// TIA Portal project "MaquinaEmbalarAut" (V14)
// Automated Packaging Machine Using PLC

(* hardware
DEVICE "S7-1200 station_1"  S7-1200 Station
   slot 0: "Rack_0"  S7-1200 Rack  Rack  V1.0
   slot 1: "Embaladora automatica"  CPU 1214C DC/DC/DC  6ES7 214-1AG40-0XB0  V4.2
*)

// ===== PLC "Embaladora automatica"  CPU 1214C DC/DC/DC =====

VAR_GLOBAL   // PLC tag table "Default tag table"
   "System_Byte" AT %MB0 : Byte;
   "FirstScan" AT %M0.0 : Bool;
   "DiagStatusUpdate" AT %M0.1 : Bool;
   "AlwaysTRUE" AT %M0.2 : Bool;
   "AlwaysFALSE" AT %M0.3 : Bool;
   "Clock_Byte" AT %MB1 : Byte;
   "Clock_10Hz" AT %M1.0 : Bool;
   "Clock_5Hz" AT %M1.1 : Bool;
   "Clock_2.5Hz" AT %M1.2 : Bool;
   "Clock_2Hz" AT %M1.3 : Bool;
   "Clock_1.25Hz" AT %M1.4 : Bool;
   "Clock_1Hz" AT %M1.5 : Bool;
   "Clock_0.625Hz" AT %M1.6 : Bool;
   "Clock_0.5Hz" AT %M1.7 : Bool;
   "LigaEsteiraCaixa" AT %M10.0 : Bool;
   "LigaEsteiraProdutos" AT %M20.0 : Bool;
   "Zera cont" AT %M100.5 : Bool;
END_VAR

VAR_GLOBAL   // PLC tag table "Inputs"
   "SensorProduto" AT %I0.0 : Bool;
   "SensorCaixa" AT %I0.1 : Bool;
   "ChaveOnOff" AT %I0.2 : Bool;
END_VAR

VAR_GLOBAL   // PLC tag table "Outputs"
   "MotorEsteiraCaixa" AT %Q0.0 : Bool;
   "MotorEsteiraProduto" AT %Q0.1 : Bool;
   "LuzVerde" AT %Q0.2 : Bool;
   "LuzAmarela" AT %Q0.3 : Bool;
   "LuzVermelha" AT %Q0.4 : Bool;
END_VAR

DATA_BLOCK "embalados"   // DB1
{ S7_Optimized_Access := 'TRUE' }
VERSION : 0.1
   VAR
      Qembalados : Int;
   END_VAR
BEGIN
END_DATA_BLOCK

// folder: System blocks/Program resources

DATA_BLOCK "IEC_Counter_0_DB"   // DB2
{ S7_Optimized_Access := 'TRUE' }
AUTHOR : Simatic
FAMILY : IEC
NAME : CNTR
VERSION : 1.0
// stored: InstanceOfName IEC_COUNTER
"IEC_COUNTER"
BEGIN
END_DATA_BLOCK

// folder: (top level)

FUNCTION "Outputs" : Void   // FC1, LAD
{ S7_Optimized_Access := 'TRUE' }
VERSION : 0.1
BEGIN

REGION Network 1: "MotorEsteiraCaixa"
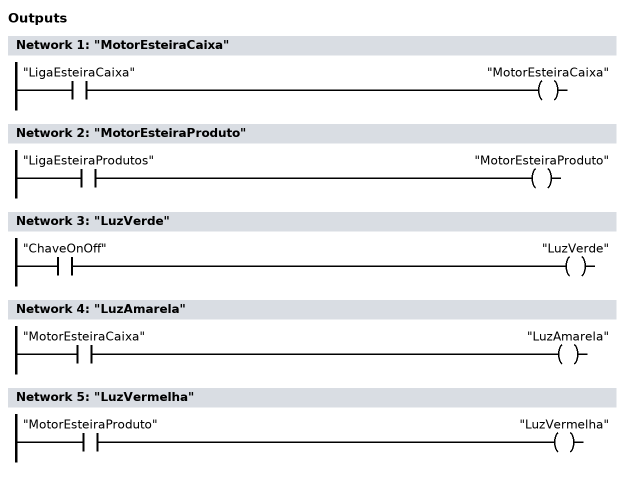
   RUNG wire#powerrail
      Contact( "LigaEsteiraCaixa" )
      Coil( "MotorEsteiraCaixa" )
   END_RUNG
   // the same network as SCL:
   "MotorEsteiraCaixa" := "LigaEsteiraCaixa";
END_REGION

REGION Network 2: "MotorEsteiraProduto"
   RUNG wire#powerrail
      Contact( "LigaEsteiraProdutos" )
      Coil( "MotorEsteiraProduto" )
   END_RUNG
   // the same network as SCL:
   "MotorEsteiraProduto" := "LigaEsteiraProdutos";
END_REGION

REGION Network 3: "LuzVerde"
   RUNG wire#powerrail
      Contact( "ChaveOnOff" )
      Coil( "LuzVerde" )
   END_RUNG
   // the same network as SCL:
   "LuzVerde" := "ChaveOnOff";
END_REGION

REGION Network 4: "LuzAmarela"
   RUNG wire#powerrail
      Contact( "MotorEsteiraCaixa" )
      Coil( "LuzAmarela" )
   END_RUNG
   // the same network as SCL:
   "LuzAmarela" := "MotorEsteiraCaixa";
END_REGION

REGION Network 5: "LuzVermelha"
   RUNG wire#powerrail
      Contact( "MotorEsteiraProduto" )
      Coil( "LuzVermelha" )
   END_RUNG
   // the same network as SCL:
   "LuzVermelha" := "MotorEsteiraProduto";
END_REGION
END_FUNCTION

FUNCTION "ControlEsteira" : Void   // FC2, LAD
{ S7_Optimized_Access := 'TRUE' }
VERSION : 0.1
   VAR_TEMP
      Temp_1 : Int;
   END_VAR
BEGIN

REGION Network 1: Controle Esteira Inferior Caixas
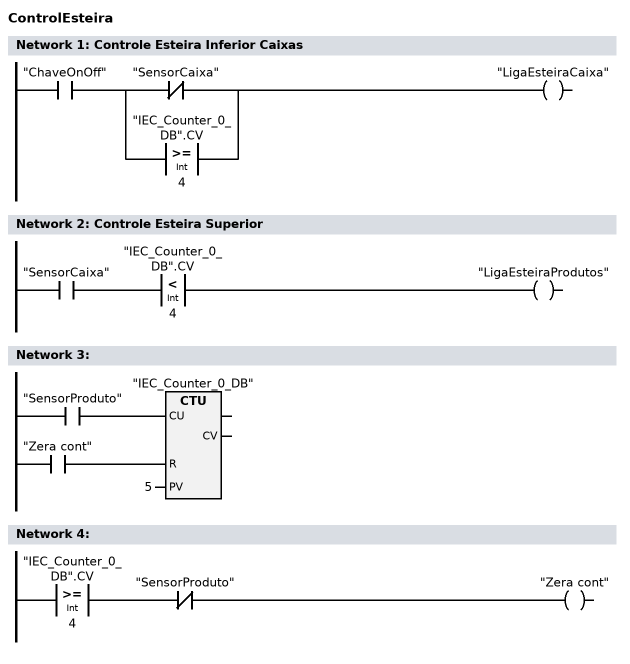
   RUNG wire#powerrail
      Contact( "ChaveOnOff" )
      wire#w1
      I_Contact( "SensorCaixa" )
      wire#w2
      Coil( "LigaEsteiraCaixa" )
   END_RUNG
   RUNG wire#w1
      { S7_Templates := "SrcType := Int" } GE_Contact(in1 := "IEC_Counter_0_DB".CV, in2 := 4)
   END_RUNG wire#w2
   // the same network as SCL:
   "LigaEsteiraCaixa" := "ChaveOnOff" AND (NOT "SensorCaixa" OR ("IEC_Counter_0_DB".CV >= 4));
END_REGION

REGION Network 2: Controle Esteira Superior
   RUNG wire#powerrail
      Contact( "SensorCaixa" )
      { S7_Templates := "SrcType := Int" } LT_Contact(in1 := "IEC_Counter_0_DB".CV, in2 := 4)
      Coil( "LigaEsteiraProdutos" )
   END_RUNG
   // the same network as SCL:
   "LigaEsteiraProdutos" := "SensorCaixa" AND ("IEC_Counter_0_DB".CV < 4);
END_REGION

REGION Network 3
   "IEC_Counter_0_DB".CTU(CU := "SensorProduto", R := "Zera cont", PV := 5);
END_REGION

REGION Network 4
   RUNG wire#powerrail
      { S7_Templates := "SrcType := Int" } GE_Contact(in1 := "IEC_Counter_0_DB".CV, in2 := 4)
      I_Contact( "SensorProduto" )
      Coil( "Zera cont" )
   END_RUNG
   // the same network as SCL:
   "Zera cont" := ("IEC_Counter_0_DB".CV >= 4) AND NOT "SensorProduto";
END_REGION
END_FUNCTION

ORGANIZATION_BLOCK "Main"   // OB1, LAD, ProgramCycle
TITLE = "Main Program Sweep (Cycle)"
{ S7_Optimized_Access := 'TRUE' }
VERSION : 0.1
   VAR_INPUT
      Initial_Call : Bool;   // Initial call of this OB
      Remanence : Bool;   // =True, if remanent data are available
   END_VAR
BEGIN

REGION Network 1
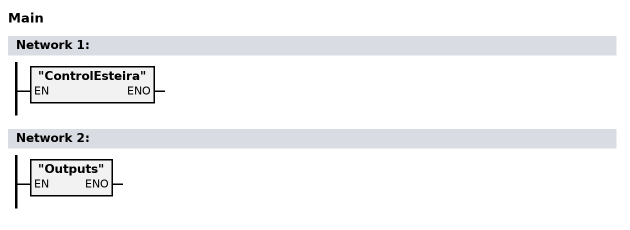
   RUNG wire#powerrail
      "ControlEsteira"()
   END_RUNG
   // the same network as SCL:
   "ControlEsteira"();
END_REGION

REGION Network 2
   RUNG wire#powerrail
      "Outputs"()
   END_RUNG
   // the same network as SCL:
   "Outputs"();
END_REGION
END_ORGANIZATION_BLOCK